(* Schneider Machine Expert - Basic project SISTEMA DE LIMPEZA DE PECAS, file version 2.7.0.0 *)
(* ProjectInformations: Name=Novo projeto *)

HARDWARE
  Cpu 0: TM221CE40R
  EthernetConfiguration: NetworkName=M221, IpAllocationMode=FixedAddress, IpAddress=0.0.0.0, SubnetMask=0.0.0.0
  SerialLineConfiguration: Baud=Baud19200, Parity=ParityEven, DataBits=DataBits8, StopBits=StopBits1, PhysicalMedium=PhysicalMediumRs485, TransmissionMode=TransmissionModeModbusRtu, SlaveId=1, Addressing=SlaveAddressing
  MastTask: UsePeriodScanMode=false, PeriodScan=100
  FastTask: Period=255
  CpuBehavior: StartingMode=StartAsPreviousState, AutoSaveRamOnEeprom=true, WatchdogPeriod=250

SYMBOLS  (address, symbol, comment, settings)
  %M0       FS  "FIRST SCAN"
  %M1       CRT_FS  "CORTA FIRST SCAN"
  %M2       PASSO_0  "CONDIÇÃO INICIAL"
  %M3       PASSO_1  "SUBIR TALHA"
  %M4       PASSO_2  "LEVAR TALHA PARA DIREITA"
  %M5       PASSO_3  "ESPERAR 10s E DESCER TALHA"
  %M6       PASSO_4  "ESPERAR 30s E SUBIR TALHA"
  %M7       PASSO_5  "LEVAR TALHA PARA DIREITA"
  %M8       PASSO_6  "ESPERAR 10s E DESCER TALHA"
  %M9       PASSO_7  "ESPERAR 60s E SUBIR TALHA"
  %M10      M_VC_1  "MEMORIA MOTOR VERTICAL CIMA"
  %M11      M_VC_2  "MEMORIA MOTOR VERTICAL CIMA 2"
  %M12      M_VC_3  "MEMORIA MOTOR VERCIAL CIMA 3"
  %M13      M_VC_4  "MEMORIA MOTOR VERTICAL CIMA 4"
  %M14      M_HD_1  "MEMORIA MOTOR HORIZONTAL DIREITA 1"
  %M15      M_HD_2  "MEMORIA MOTOR HORIZONTAL DIREITA 2"
  %M16      M_VB_1  "MEMORIA MOTOR VERTICAL BAIXO 1"
  %M17      M_VB_2  "MEMORIA MOTOR VERTICAL BAIXO 2"
  %M18      M_VB_3  "MEMORIA MOTOR VERTICAL BAIXO 3"
  %M19      M_HE_1  "MEMORIA MOTOR HORIZONTAL ESQUERDA 1"
  %TM0      T1  "TEMPORIZADOR PARADA TALHA"  [Preset=10, Base=OneSecond]
  %TM1      T2  "TEMPORIZADOR TANQUE 1"  [Preset=30, Base=OneSecond]
  %TM2      T3  "TEMPORIZADOR TANQUE 2"  [Preset=60, Base=OneSecond]
  %I0.0     B0  "BOTÃO START"
  %I0.1     YA  "SENSOR TALHA ALTA"
  %I0.2     YB  "SENSOR TALHA BAIXA"
  %I0.3     X1  "AREA DE CARGA E DESCARGA"
  %I0.4     X2  "AREA DO TANQUE 1"
  %I0.5     X3  "AREA DO TANQUE 2"
  %Q0.0     MX_1  "MOTOR HORIZONTAL ACIONAMENTO DIREITA"
  %Q0.1     MX_2  "MOTOR HORIZONTAL ACIONAMENTO ESQUERDA"
  %Q0.2     MY_1  "MOTOR VERTICAL ACIONAMENTO CIMA"
  %Q0.3     MY_2  "MOTOR VERTICAL ACIONAMENTO BAIXO"

POU PASSOS
  (* SectionNumber=1 *)

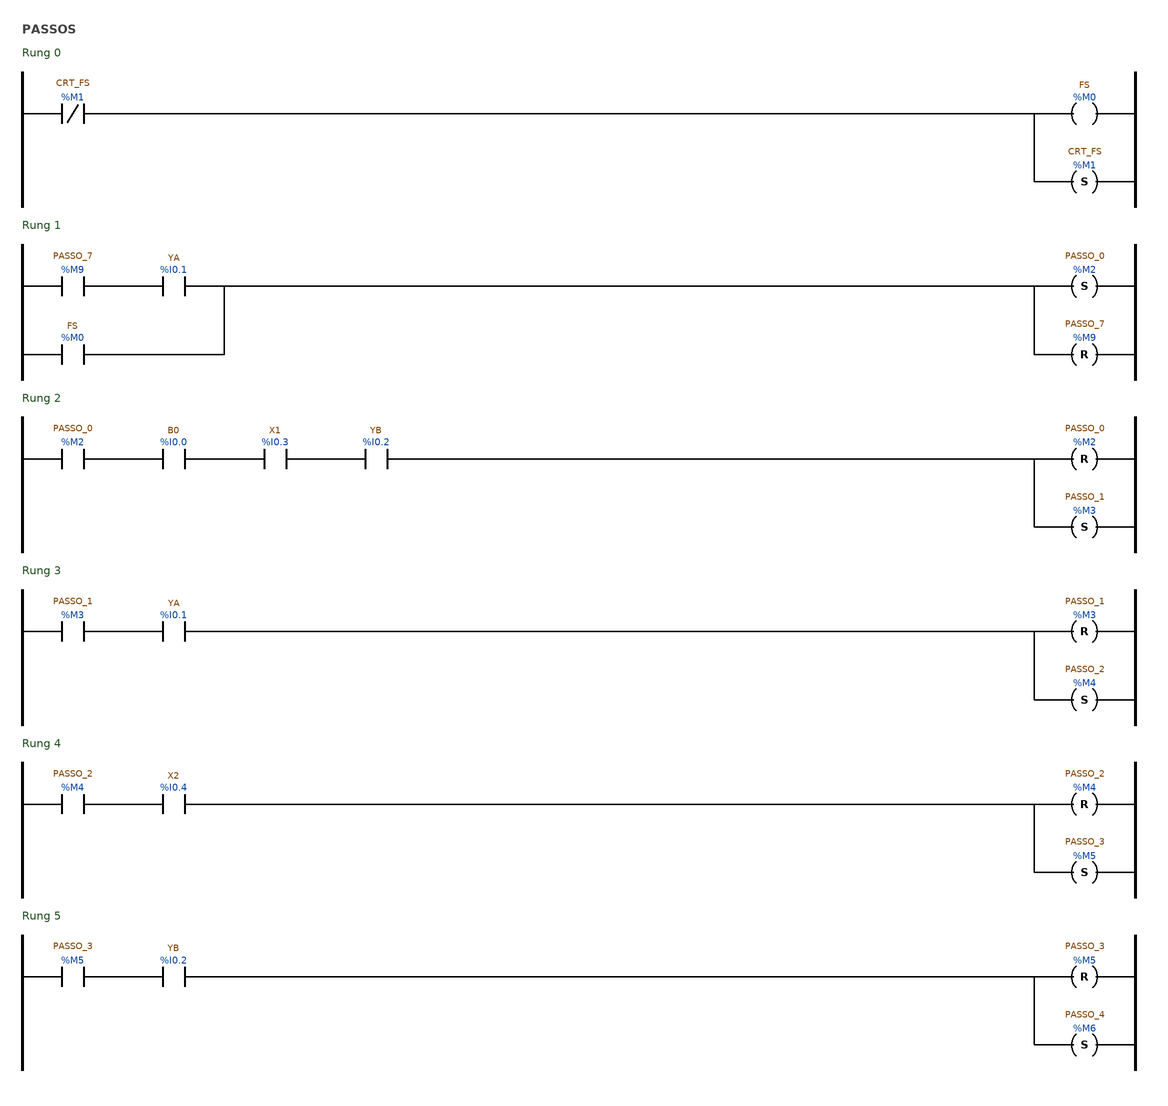

// Rung 0
  LDN %M1                 (* CRT_FS *)
  ST %M0                  (* FS *)
  S %M1                   (* CRT_FS *)
  // as ST:
  //   FS := NOT CRT_FS;
  //   IF NOT CRT_FS THEN CRT_FS := TRUE; END_IF;

// Rung 1
  LD %M9                  (* PASSO_7 *)
  AND %I0.1               (* YA *)
  OR %M0                  (* FS *)
  S %M2                   (* PASSO_0 *)
  R %M9                   (* PASSO_7 *)
  // as ST:
  //   IF PASSO_7 AND YA OR FS THEN PASSO_0 := TRUE; END_IF;
  //   IF PASSO_7 AND YA OR FS THEN PASSO_7 := FALSE; END_IF;

// Rung 2
  LD %M2                  (* PASSO_0 *)
  AND %I0.0               (* B0 *)
  AND %I0.3               (* X1 *)
  AND %I0.2               (* YB *)
  R %M2                   (* PASSO_0 *)
  S %M3                   (* PASSO_1 *)
  // as ST:
  //   _t1 := PASSO_0 AND B0 AND X1 AND YB;
  //   IF _t1 THEN PASSO_0 := FALSE; END_IF;
  //   IF _t1 THEN PASSO_1 := TRUE; END_IF;

// Rung 3
  LD %M3                  (* PASSO_1 *)
  AND %I0.1               (* YA *)
  R %M3                   (* PASSO_1 *)
  S %M4                   (* PASSO_2 *)
  // as ST:
  //   _t1 := PASSO_1 AND YA;
  //   IF _t1 THEN PASSO_1 := FALSE; END_IF;
  //   IF _t1 THEN PASSO_2 := TRUE; END_IF;

// Rung 4
  LD %M4                  (* PASSO_2 *)
  AND %I0.4               (* X2 *)
  R %M4                   (* PASSO_2 *)
  S %M5                   (* PASSO_3 *)
  // as ST:
  //   _t1 := PASSO_2 AND X2;
  //   IF _t1 THEN PASSO_2 := FALSE; END_IF;
  //   IF _t1 THEN PASSO_3 := TRUE; END_IF;

// Rung 5
  LD %M5                  (* PASSO_3 *)
  AND %I0.2               (* YB *)
  R %M5                   (* PASSO_3 *)
  S %M6                   (* PASSO_4 *)
  // as ST:
  //   _t1 := PASSO_3 AND YB;
  //   IF _t1 THEN PASSO_3 := FALSE; END_IF;
  //   IF _t1 THEN PASSO_4 := TRUE; END_IF;

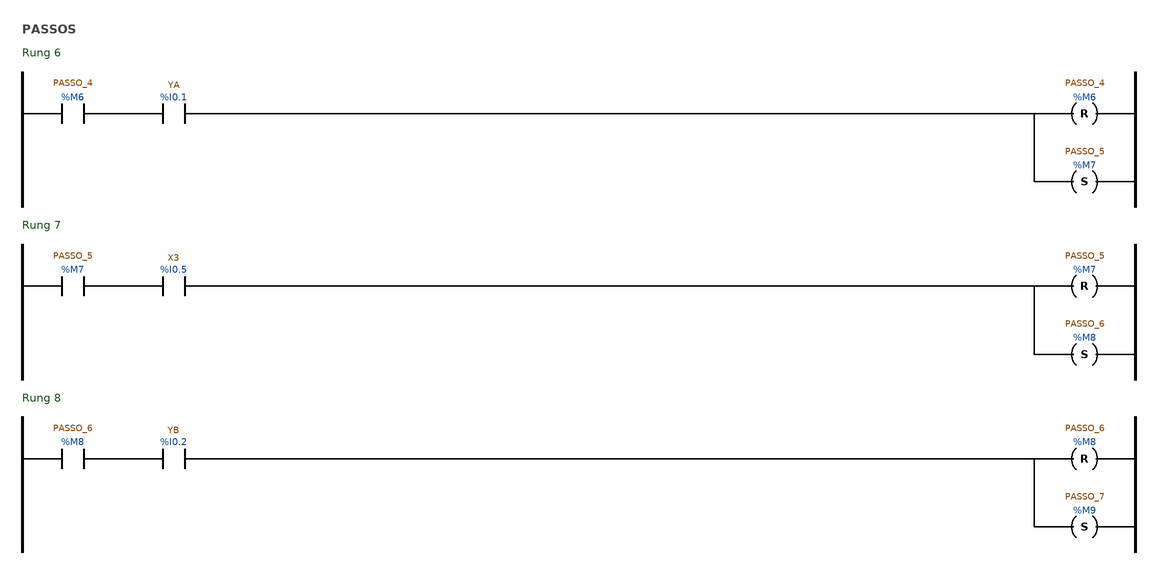

// Rung 6
  LD %M6                  (* PASSO_4 *)
  AND %I0.1               (* YA *)
  R %M6                   (* PASSO_4 *)
  S %M7                   (* PASSO_5 *)
  // as ST:
  //   _t1 := PASSO_4 AND YA;
  //   IF _t1 THEN PASSO_4 := FALSE; END_IF;
  //   IF _t1 THEN PASSO_5 := TRUE; END_IF;

// Rung 7
  LD %M7                  (* PASSO_5 *)
  AND %I0.5               (* X3 *)
  R %M7                   (* PASSO_5 *)
  S %M8                   (* PASSO_6 *)
  // as ST:
  //   _t1 := PASSO_5 AND X3;
  //   IF _t1 THEN PASSO_5 := FALSE; END_IF;
  //   IF _t1 THEN PASSO_6 := TRUE; END_IF;

// Rung 8
  LD %M8                  (* PASSO_6 *)
  AND %I0.2               (* YB *)
  R %M8                   (* PASSO_6 *)
  S %M9                   (* PASSO_7 *)
  // as ST:
  //   _t1 := PASSO_6 AND YB;
  //   IF _t1 THEN PASSO_6 := FALSE; END_IF;
  //   IF _t1 THEN PASSO_7 := TRUE; END_IF;

POU PROCESSO
  (* SectionNumber=2 *)

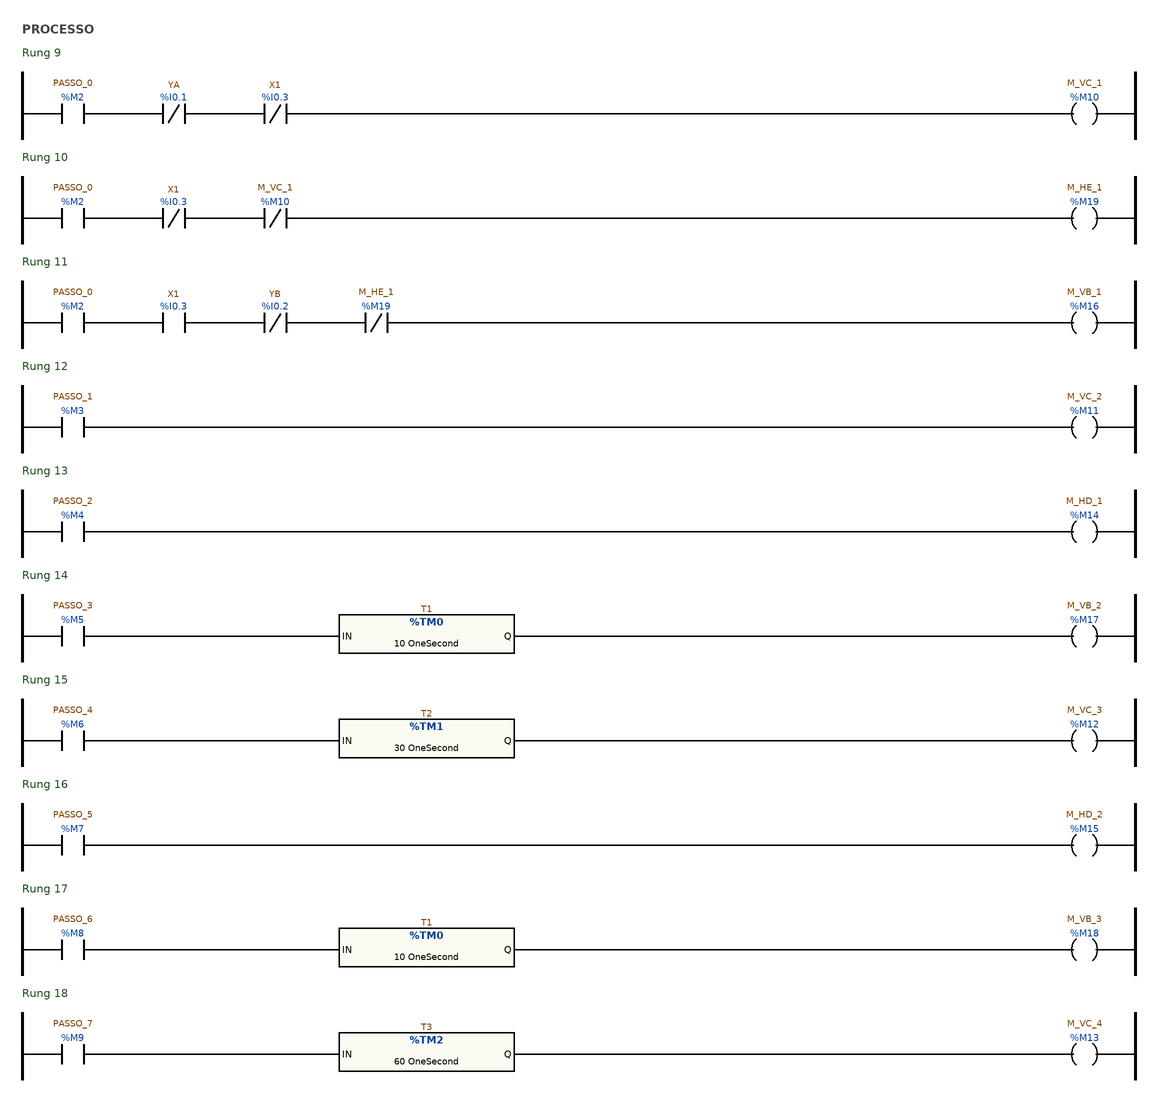

// Rung 9
  LD %M2                  (* PASSO_0 *)
  ANDN %I0.1              (* YA *)
  ANDN %I0.3              (* X1 *)
  ST %M10                 (* M_VC_1 *)
  // as ST:
  //   M_VC_1 := PASSO_0 AND NOT YA AND NOT X1;

// Rung 10
  LD %M2                  (* PASSO_0 *)
  ANDN %I0.3              (* X1 *)
  ANDN %M10               (* M_VC_1 *)
  ST %M19                 (* M_HE_1 *)
  // as ST:
  //   M_HE_1 := PASSO_0 AND NOT X1 AND NOT M_VC_1;

// Rung 11
  LD %M2                  (* PASSO_0 *)
  AND %I0.3               (* X1 *)
  ANDN %I0.2              (* YB *)
  ANDN %M19               (* M_HE_1 *)
  ST %M16                 (* M_VB_1 *)
  // as ST:
  //   M_VB_1 := PASSO_0 AND X1 AND NOT YB AND NOT M_HE_1;

// Rung 12
  LD %M3                  (* PASSO_1 *)
  ST %M11                 (* M_VC_2 *)
  // as ST:
  //   M_VC_2 := PASSO_1;

// Rung 13
  LD %M4                  (* PASSO_2 *)
  ST %M14                 (* M_HD_1 *)
  // as ST:
  //   M_HD_1 := PASSO_2;

// Rung 14
  BLK %TM0                (* T1 *)
  LD %M5                  (* PASSO_3 *)
  IN
  OUT_BLK
  LD Q
  ST %M17                 (* M_VB_2 *)
  END_BLK
  // as ST:
  //   T1(IN := PASSO_3);
  //   M_VB_2 := T1.Q;

// Rung 15
  BLK %TM1                (* T2 *)
  LD %M6                  (* PASSO_4 *)
  IN
  OUT_BLK
  LD Q
  ST %M12                 (* M_VC_3 *)
  END_BLK
  // as ST:
  //   T2(IN := PASSO_4);
  //   M_VC_3 := T2.Q;

// Rung 16
  LD %M7                  (* PASSO_5 *)
  ST %M15                 (* M_HD_2 *)
  // as ST:
  //   M_HD_2 := PASSO_5;

// Rung 17
  BLK %TM0                (* T1 *)
  LD %M8                  (* PASSO_6 *)
  IN
  OUT_BLK
  LD Q
  ST %M18                 (* M_VB_3 *)
  END_BLK
  // as ST:
  //   T1(IN := PASSO_6);
  //   M_VB_3 := T1.Q;

// Rung 18
  BLK %TM2                (* T3 *)
  LD %M9                  (* PASSO_7 *)
  IN
  OUT_BLK
  LD Q
  ST %M13                 (* M_VC_4 *)
  END_BLK
  // as ST:
  //   T3(IN := PASSO_7);
  //   M_VC_4 := T3.Q;

POU SAIDAS
  (* SectionNumber=3 *)

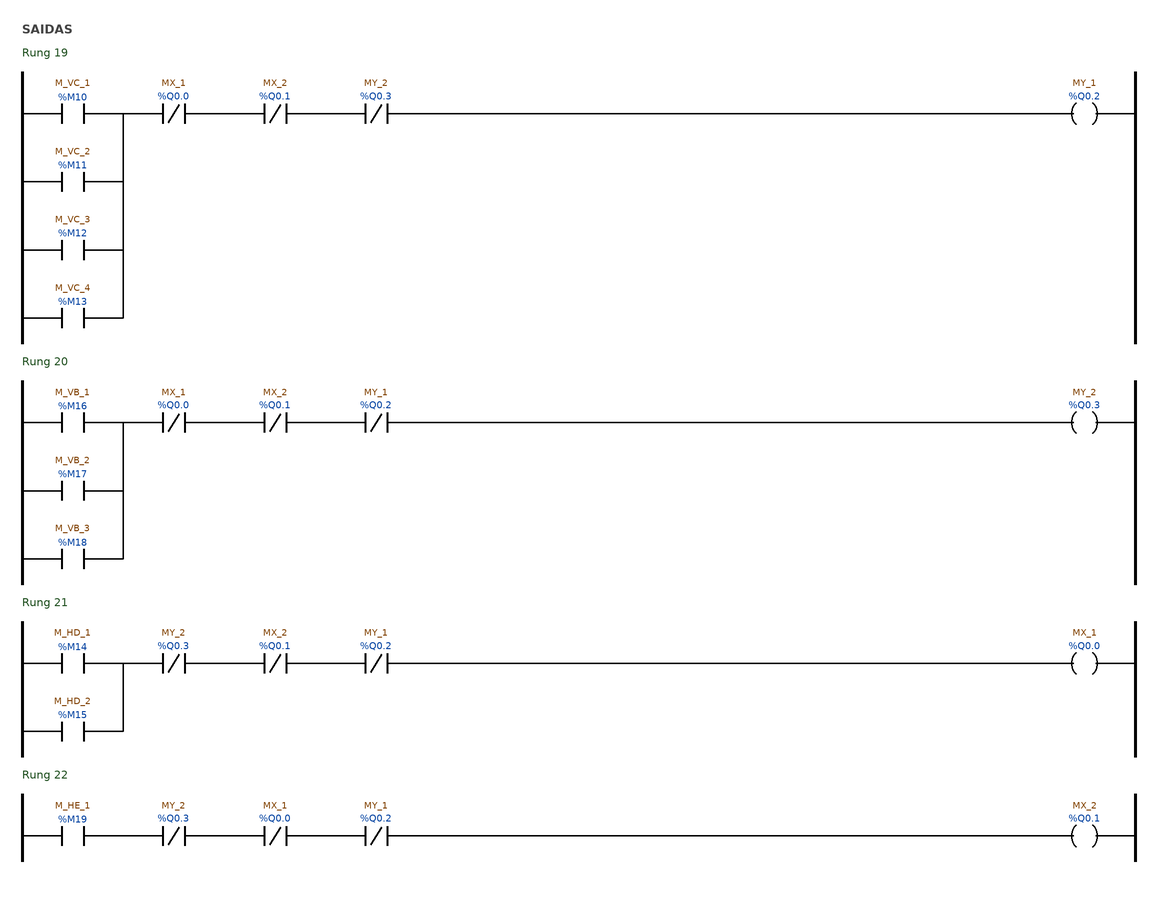

// Rung 19
  LD %M10                 (* M_VC_1 *)
  OR %M11                 (* M_VC_2 *)
  OR %M12                 (* M_VC_3 *)
  OR %M13                 (* M_VC_4 *)
  ANDN %Q0.0              (* MX_1 *)
  ANDN %Q0.1              (* MX_2 *)
  ANDN %Q0.3              (* MY_2 *)
  ST %Q0.2                (* MY_1 *)
  // as ST:
  //   MY_1 := (M_VC_1 OR M_VC_2 OR M_VC_3 OR M_VC_4) AND NOT MX_1 AND NOT MX_2 AND NOT MY_2;

// Rung 20
  LD %M16                 (* M_VB_1 *)
  OR %M17                 (* M_VB_2 *)
  OR %M18                 (* M_VB_3 *)
  ANDN %Q0.0              (* MX_1 *)
  ANDN %Q0.1              (* MX_2 *)
  ANDN %Q0.2              (* MY_1 *)
  ST %Q0.3                (* MY_2 *)
  // as ST:
  //   MY_2 := (M_VB_1 OR M_VB_2 OR M_VB_3) AND NOT MX_1 AND NOT MX_2 AND NOT MY_1;

// Rung 21
  LD %M14                 (* M_HD_1 *)
  OR %M15                 (* M_HD_2 *)
  ANDN %Q0.3              (* MY_2 *)
  ANDN %Q0.1              (* MX_2 *)
  ANDN %Q0.2              (* MY_1 *)
  ST %Q0.0                (* MX_1 *)
  // as ST:
  //   MX_1 := (M_HD_1 OR M_HD_2) AND NOT MY_2 AND NOT MX_2 AND NOT MY_1;

// Rung 22
  LD %M19                 (* M_HE_1 *)
  ANDN %Q0.3              (* MY_2 *)
  ANDN %Q0.0              (* MX_1 *)
  ANDN %Q0.2              (* MY_1 *)
  ST %Q0.1                (* MX_2 *)
  // as ST:
  //   MX_2 := M_HE_1 AND NOT MY_2 AND NOT MX_1 AND NOT MY_1;
